// TIA Portal project "FB_Bedienpult" (V20)

(* hardware
DEVICE "S7-1500/ET200MP-Station_1"  S7-1500 station
   slot 0: "Profilschiene_0"  Rack  6ES7 590-1***0-0AA0
   slot 1: "PLC_1"  CPU 1513-1 PN  6ES7 513-1AM03-0AB0  V4.0
      slot 3: "CPU-Display_1"  6ES7591-1AA00-0AA0
      slot 32768: "PROFINET-Schnittstelle_1"  X1
         slot 32769: "Port_1"  X1 P1
         slot 32770: "Port_2"  X1 P2
      slot 34817: "Virtual CP interface port_1"  Virtual CP interface port  Virtual CP interface port FW V4.0
   slot 2: "DI 16x24VDC BA_1"  DI 16x24VDC BA  6ES7 521-1BH10-0AA0  V1.1
   slot 3: "DQ 16x24VDC/0.5A ST_1"  DQ 16x24VDC/0.5A ST  6ES7 522-1BH00-0AB0  V2.0
   slot 4: "AI 8xU/I/R/RTD BA_2"  AI 8xU/I/R/RTD BA  6ES7 531-7QF00-0AB0  V1.0
   slot 5: "AQ 8xU/I HS_2"  AQ 8xU/I HS  6ES7 532-5HF00-0AB0  V2.2
*)

// ===== PLC "PLC_1"  CPU 1513-1 PN =====

VAR_GLOBAL   // PLC tag table "Standard-Variablentabelle"
   "Clock_Byte" AT %MB0 : Byte;
   "Clock_10Hz" AT %M0.0 : Bool;
   "Clock_5Hz" AT %M0.1 : Bool;
   "Clock_2.5Hz" AT %M0.2 : Bool;
   "Clock_2Hz" AT %M0.3 : Bool;
   "Clock_1.25Hz" AT %M0.4 : Bool;
   "Clock_1Hz" AT %M0.5 : Bool;
   "Clock_0.625Hz" AT %M0.6 : Bool;
   "Clock_0.5Hz" AT %M0.7 : Bool;
END_VAR

VAR_GLOBAL   // PLC tag table "Ausgaenge"
   "H1" AT %Q0.1 : Bool;   // Meldeleuchte (Start)
   "H2" AT %Q0.2 : Bool;   // Meldeleuchte (Stopp)
   "H3" AT %Q0.3 : Bool;   // Meldeleuchte (Reset)
END_VAR

VAR_GLOBAL   // PLC tag table "Eingaenge"
   "S0" AT %I0.0 : Bool;   // Not-Aus
   "S1" AT %I0.1 : Bool;   // Starttaster
   "S2" AT %I0.2 : Bool;   // Stopptaster
   "S3" AT %I0.3 : Bool;   // Resettaster
END_VAR

DATA_BLOCK "Anlagensteuerung_DB"   // DB1
{ S7_Optimized_Access := 'TRUE' }
VERSION : 0.1
// stored: InstanceOfName Anlagensteuerung
"Anlagensteuerung"
BEGIN
END_DATA_BLOCK

DATA_BLOCK "Bedienpult_DB"   // DB2
{ S7_Optimized_Access := 'TRUE' }
VERSION : 0.1
// stored: InstanceOfName Bedienpult
"Bedienpult"
BEGIN
END_DATA_BLOCK

FUNCTION_BLOCK "Anlagensteuerung"   // FB1, FBD
{ S7_Optimized_Access := 'TRUE' }
VERSION : 0.1
   VAR_INPUT
      "Not-Aus" : Bool;
      Start : Bool;
      Stopp : Bool;
      Reset : Bool;
   END_VAR
   VAR_OUTPUT
      NotAus_aktiv : Bool;
      Anlage_aktiv : Bool;
   END_VAR
   VAR
      Merker_NotAus_aktiv : Bool;
      Merker_Anlage_aktiv : Bool;
   END_VAR
BEGIN

REGION Network 1
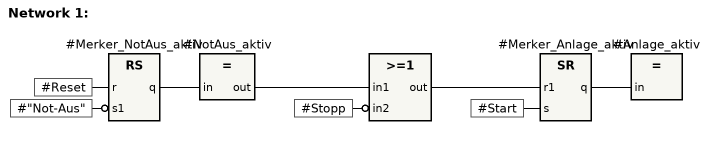
   IF #Reset THEN
       #Merker_NotAus_aktiv := FALSE;   // RS flip-flop
   END_IF;
   IF NOT #"Not-Aus" THEN #Merker_NotAus_aktiv := TRUE; END_IF;
   #NotAus_aktiv := #Merker_NotAus_aktiv;
   IF #Start THEN
       #Merker_Anlage_aktiv := TRUE;   // SR flip-flop
   END_IF;
   IF #Merker_NotAus_aktiv OR NOT #Stopp THEN #Merker_Anlage_aktiv := FALSE; END_IF;
   #Anlage_aktiv := #Merker_Anlage_aktiv;
END_REGION
END_FUNCTION_BLOCK

FUNCTION_BLOCK "Bedienpult"   // FB2, FBD
{ S7_Optimized_Access := 'TRUE' }
VERSION : 0.1
   VAR_INPUT
      NotAus_Schalter : Bool;
      Start_Taster : Bool;
      Stop_Taster : Bool;
      Reset_Taster : Bool;
      Taktmerker : Bool;
   END_VAR
   VAR_OUTPUT
      NotAus_aktiv : Bool;
      AnlageEin_aktiv : Bool;
      Meldeleuchte_gruen : Bool;
      Meldleuchte_rot : Bool;
      Meldeleuchte_Reset : Bool;
   END_VAR
BEGIN

REGION Network 1
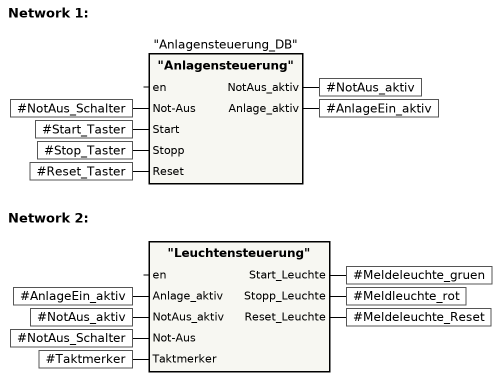
   "Anlagensteuerung_DB"("Not-Aus" := #NotAus_Schalter,   // "Anlagensteuerung"
                         Start := #Start_Taster,
                         Stopp := #Stop_Taster,
                         Reset := #Reset_Taster,
                         NotAus_aktiv => #NotAus_aktiv,
                         Anlage_aktiv => #AnlageEin_aktiv);
END_REGION

REGION Network 2
   "Leuchtensteuerung"(Anlage_aktiv := #AnlageEin_aktiv,
                       NotAus_aktiv := #NotAus_aktiv,
                       "Not-Aus" := #NotAus_Schalter,
                       Taktmerker := #Taktmerker,
                       Start_Leuchte => #Meldeleuchte_gruen,
                       Stopp_Leuchte => #Meldleuchte_rot,
                       Reset_Leuchte => #Meldeleuchte_Reset);
END_REGION
END_FUNCTION_BLOCK

FUNCTION "Leuchtensteuerung" : Void   // FC1, FBD
{ S7_Optimized_Access := 'TRUE' }
VERSION : 0.1
   VAR_INPUT
      Anlage_aktiv : Bool;
      NotAus_aktiv : Bool;
      "Not-Aus" : Bool;
      Taktmerker : Bool;
   END_VAR
   VAR_OUTPUT
      Start_Leuchte : Bool;
      Stopp_Leuchte : Bool;
      Reset_Leuchte : Bool;
   END_VAR
BEGIN

REGION Network 1
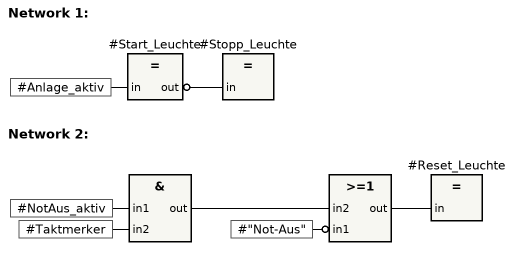
   #Start_Leuchte := #Anlage_aktiv;
   #Stopp_Leuchte := NOT #Anlage_aktiv;
END_REGION

REGION Network 2
   #Reset_Leuchte := (#NotAus_aktiv AND #Taktmerker) OR NOT #"Not-Aus";
END_REGION
END_FUNCTION

ORGANIZATION_BLOCK "Main"   // OB1, FBD, ProgramCycle
TITLE = "Main Program Sweep (Cycle)"
{ S7_Optimized_Access := 'TRUE' }
VERSION : 0.1
   VAR_INPUT
      Initial_Call : Bool;   // Initial call of this OB
      Remanence : Bool;   // =True, if remanent data are available
   END_VAR
BEGIN

REGION Network 1
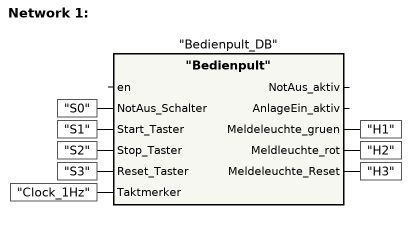
   "Bedienpult_DB"(NotAus_Schalter := "S0",   // "Bedienpult"
                   Start_Taster := "S1",
                   Stop_Taster := "S2",
                   Reset_Taster := "S3",
                   Taktmerker := "Clock_1Hz",
                   Meldeleuchte_gruen => "H1",
                   Meldleuchte_rot => "H2",
                   Meldeleuchte_Reset => "H3");
END_REGION
END_ORGANIZATION_BLOCK